# EPICS autosave request: iocBoot/ioc13cygwin/auto_settings.req
file "ccd_settings.req",                P=13Cygwin:, C=ccd1
file "scan_settings.req",               P=13Cygwin:, S=scan1
file "scan_settings.req",               P=13Cygwin:, S=scan2
file "scan_settings.req",               P=13Cygwin:, S=scan3
file "scan_settings.req",               P=13Cygwin:, S=scan4
file "CARS_motor_settings.req",         P=13Cygwin:, M=m1
file "CARS_motor_settings.req",         P=13Cygwin:, M=m2
file "CARS_motor_settings.req",         P=13Cygwin:, M=m3
